FUNCTION_BLOCK HandshakeResponder (* Handshake pattern demo: Socket / Responder role *)
  (* Standard: 61499-2; Description: Copyright (c) 2026 Meisterschulen am Ostbahnhof This program and the accompanying materials are made available under the terms of the Eclipse Public License 2.0 which is available at https://www.eclipse.org/legal/epl-2.0/ SPDX-License-Identifier: EPL-2.0 *)
  (* Version 1.3, 2026-08-31, Franz Höpfinger, Meisterschulen am Ostbahnhof, Fixed INIT handling: dedicated Init/Initialized/DeInit states with INIT[TRUE=QI]/INIT[FALSE=QI] guards (per TemplateBasic.fbt), instead of resetting counters on every re-entry to idle *)
  (* Version 1.2, 2026-08-31, Franz Höpfinger, Meisterschulen am Ostbahnhof, EVENT_HS EventInputs/EventOutputs swapped so the Responder is now a Socket (more natural layout) - back to Sockets here *)
  (* Version 1.1, 2026-08-31, Franz Höpfinger, Meisterschulen am Ostbahnhof, Handshake design pattern (IEC 61499 primer course, Module 6, Valeriy Vyatkin), demo Responder *)
  (* Version 1.0, 2026-08-31, Franz Höpfinger, Meisterschulen am Ostbahnhof, initial version, wrongly declared as Socket - fixed to Plug *)
  PACKAGE Meins::DesingPatterns::HandshakePattern;
  (* Documentation:
  Responder ("server") side of the Handshake design pattern (IEC 61499 primer course, Module 6, Valeriy Vyatkin, slide 72).
   Uses the dataless adapter::events::Handshake::EVENT_HS adapter as a Socket: receives REQ and answers with CNF; on TRIGGER it sends an unsolicited IND and counts the matching RSP once the Requester acknowledges it.
   Per the adapter's own declaration, the Socket side is the one that fires CNF/IND and reacts to REQ/RSP - i.e. the Socket plays the server/Responder role here, the Plug plays the client/Requester role. See HandshakePattern.md in this folder for the full write-up.
  *)
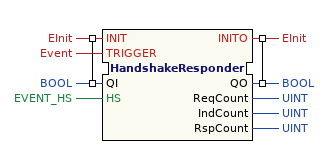
  EVENT_INPUT
    INIT : EInit WITH QI; (* Initialization Request *)
    TRIGGER; (* Demo: fire an unsolicited IND towards the Requester *)
  END_EVENT
  EVENT_OUTPUT
    INITO : EInit WITH QO; (* Initialization Confirm *)
  END_EVENT
  VAR_INPUT
    QI : BOOL; (* Input event qualifier *)
  END_VAR
  VAR_OUTPUT
    QO : BOOL; (* Output event qualifier *)
    ReqCount : UINT; (* Number of REQ received (demo counter) *)
    IndCount : UINT; (* Number of IND sent (demo counter) *)
    RspCount : UINT; (* Number of RSP received (demo counter) *)
  END_VAR
  SOCKETS
    HS : adapter::events::Handshake::EVENT_HS; (* Handshake socket: receives REQ/RSP, emits CNF/IND *)
  END_SOCKETS
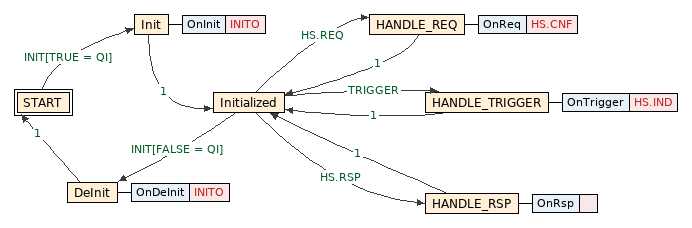
  EC_STATES
    START; (* Uninitialized *)
    Init : OnInit -> INITO; (* Initialization *)
    Initialized; (* Idle, ready to react *)
    DeInit : OnDeInit -> INITO; (* De-initialization *)
    HANDLE_REQ : OnReq -> HS.CNF; (* Answer a REQ with CNF *)
    HANDLE_TRIGGER : OnTrigger -> HS.IND; (* Send an unsolicited IND *)
    HANDLE_RSP : OnRsp; (* Acknowledge an RSP *)
  END_STATES
  EC_TRANSITIONS
    START TO Init := INIT[TRUE = QI];
    Init TO Initialized := 1;
    Initialized TO DeInit := INIT[FALSE = QI];
    DeInit TO START := 1;
    Initialized TO HANDLE_REQ := HS.REQ;
    HANDLE_REQ TO Initialized := 1;
    Initialized TO HANDLE_TRIGGER := TRIGGER;
    HANDLE_TRIGGER TO Initialized := 1;
    Initialized TO HANDLE_RSP := HS.RSP;
    HANDLE_RSP TO Initialized := 1;
  END_TRANSITIONS
  ALGORITHM OnInit IN ST: (* Reset demo counters *)
ReqCount := 0;
IndCount := 0;
RspCount := 0;
QO := QI;
  END_ALGORITHM
  ALGORITHM OnDeInit IN ST: (* De-initialize *)
QO := FALSE;
  END_ALGORITHM
  ALGORITHM OnReq IN ST: (* Count a received REQ *)
ReqCount := ReqCount + 1;
  END_ALGORITHM
  ALGORITHM OnTrigger IN ST: (* Count an IND about to be sent *)
IndCount := IndCount + 1;
  END_ALGORITHM
  ALGORITHM OnRsp IN ST: (* Count a received RSP *)
RspCount := RspCount + 1;
  END_ALGORITHM
END_FUNCTION_BLOCK
